ABB RAPID module: Module1.mod

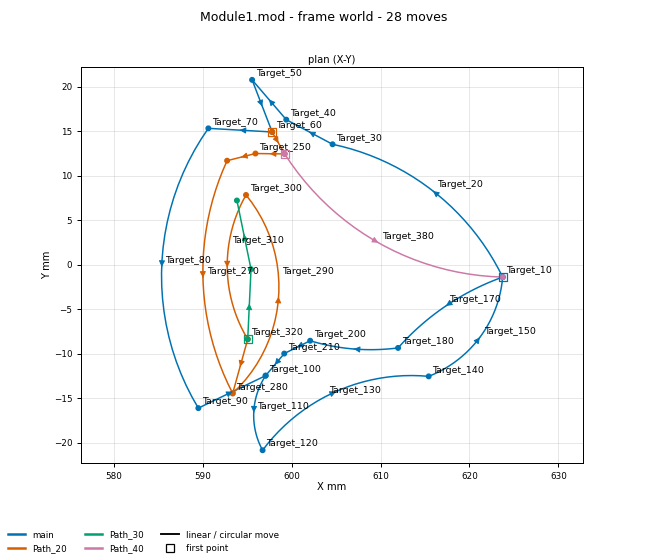
[picture p0: tool path of Module1.mod in frame world, 28 of 28 moves have a stored position in this frame; points joined in program order, loops and branches not executed]
MODULE Module1
	CONST robtarget Target_10:=[[623.736,-1.4,500],[0,0.847722968,-0.530439224,0],[-1,0,-2,0],[-1,-1,-1,-1,-1,-1]];
	CONST robtarget Target_20:=[[615.902873443,8.281748692,500],[0,0.94557602,-0.325401277,0],[0,0,-2,0],[-1,-1,-1,-1,-1,-1]];
	CONST robtarget Target_30:=[[604.61,13.532,500],[0,0.994622428,-0.103567489,0],[0,0,-2,0],[-1,-1,-1,-1,-1,-1]];
	CONST robtarget Target_40:=[[599.403600487,16.302277668,500],[0,0.943554709,-0.331216713,0],[0,0,-2,0],[-1,-1,-1,-1,-1,-1]];
	CONST robtarget Target_50:=[[595.562,20.777,500],[0,0.865930359,-0.500164587,0],[0,0,-2,0],[-1,-1,-1,-1,-1,-1]];
	CONST robtarget Target_60:=[[597.816370005,14.915141124,500],[0,0.852892303,-0.522086888,0],[0,0,-2,0],[-1,-1,-1,-1,-1,-1]];
	CONST robtarget Target_70:=[[590.643,15.324,500],[0,0.99985512,0.017021701,0],[0,0,1,0],[-1,-1,-1,-1,-1,-1]];
	CONST robtarget Target_80:=[[585.395347846,-0.237449737,500],[0,0.719631545,0.694356133,0],[-1,0,1,0],[-1,-1,-1,-1,-1,-1]];
	CONST robtarget Target_90:=[[589.518,-16.134,500],[0,0.491466316,0.870896584,0],[-1,0,0,0],[-1,-1,-1,-1,-1,-1]];
	CONST robtarget Target_100:=[[597.083,-12.483,500],[0,-0.264785252,0.964307405,0],[-1,0,-1,0],[-1,-1,-1,-1,-1,-1]];
	CONST robtarget Target_110:=[[595.746657937,-16.629604656,500],[0,0.721325087,0.69259665,0],[-1,0,1,0],[-1,-1,-1,-1,-1,-1]];
	CONST robtarget Target_120:=[[596.742,-20.871,500],[0,0.509480024,0.860482484,0],[-1,0,0,0],[-1,-1,-1,-1,-1,-1]];
	CONST robtarget Target_130:=[[603.809791295,-14.83880817,500],[0,-0.23193219,0.972731957,0],[-1,0,-1,0],[-1,-1,-1,-1,-1,-1]];
	CONST robtarget Target_140:=[[615.416517972,-12.563275607,500],[0,-0.185133559,0.982713369,0],[-1,0,-1,0],[-1,-1,-1,-1,-1,-1]];
	CONST robtarget Target_150:=[[621.175011199,-8.173115177,500],[0,-0.448574398,0.893745495,0],[-1,0,-1,0],[-1,-1,-1,-1,-1,-1]];
	CONST robtarget Target_160:=[[623.736,-1.4,500],[0,-0.677333099,0.735676473,0],[-1,0,-1,0],[-1,-1,-1,-1,-1,-1]];
	CONST robtarget Target_170:=[[617.31311623,-4.669496623,500],[0,0.926848335,0.375435965,0],[-1,0,1,0],[-1,-1,-1,-1,-1,-1]];
	CONST robtarget Target_180:=[[611.975614607,-9.363781001,500],[0,0.989682936,0.143274863,0],[-1,0,1,0],[-1,-1,-1,-1,-1,-1]];
	CONST robtarget Target_190:=[[608.374,-9.557,500],[0,0.995937158,-0.090050974,0],[-1,0,-2,0],[-1,-1,-1,-1,-1,-1]];
	CONST robtarget Target_200:=[[602.090461719,-8.557904909,500],[0,0.991973762,0.126443879,0],[-1,0,1,0],[-1,-1,-1,-1,-1,-1]];
	CONST robtarget Target_210:=[[599.177398091,-9.998243918,500],[0,0.945259462,0.326319705,0],[-1,0,1,0],[-1,-1,-1,-1,-1,-1]];
	CONST robtarget Target_220:=[[597.083,-12.483,500],[0,0.858718949,0.512446843,0],[-1,0,1,0],[-1,-1,-1,-1,-1,-1]];
	CONST robtarget Target_230:=[[597.816370005,14.915141124,500],[0,0.522086888,0.852892303,0],[0,0,0,0],[-1,-1,-1,-1,-1,-1]];
	CONST robtarget Target_240:=[[599.228158361,12.447628134,500],[0,0.481013467,0.876713205,0],[0,0,0,0],[-1,-1,-1,-1,-1,-1]];
	CONST robtarget Target_250:=[[595.93940711,12.49384908,500],[0,0.998290636,0.058444905,0],[0,0,1,0],[-1,-1,-1,-1,-1,-1]];
	CONST robtarget Target_260:=[[592.751,11.687,500],[0,0.98212196,0.18824573,0],[0,0,1,0],[-1,-1,-1,-1,-1,-1]];
	CONST robtarget Target_270:=[[590.032529197,-1.465300629,500],[0,0.698569925,0.715541794,0],[-1,0,0,0],[-1,-1,-1,-1,-1,-1]];
	CONST robtarget Target_280:=[[593.379,-14.472,500],[0,0.518908028,0.854830076,0],[-1,0,0,0],[-1,-1,-1,-1,-1,-1]];
	CONST robtarget Target_290:=[[598.550160299,-1.525622572,500],[0,0.710484728,-0.70371262,0],[-1,0,-2,0],[-1,-1,-1,-1,-1,-1]];
	CONST robtarget Target_300:=[[594.878216801,7.831632395,500],[0,0.996886245,0.078853123,0],[0,0,1,0],[-1,-1,-1,-1,-1,-1]];
	CONST robtarget Target_310:=[[592.899123752,1.965756689,500],[0,0.725029605,0.688717701,0],[0,0,1,0],[-1,-1,-1,-1,-1,-1]];
	CONST robtarget Target_320:=[[595.07,-8.388,500],[0,0.525278576,0.850930325,0],[-1,0,0,0],[-1,-1,-1,-1,-1,-1]];
	CONST robtarget Target_330:=[[593.379,-14.472,500],[0,0.825320138,0.564665096,0],[-1,0,1,0],[-1,-1,-1,-1,-1,-1]];
	CONST robtarget Target_340:=[[595.069954295,-8.387992086,500],[0,-0.64397045,0.765050364,0],[-1,0,-1,0],[-1,-1,-1,-1,-1,-1]];
	CONST robtarget Target_350:=[[595.439579744,-0.511504022,500],[0,0.734022523,-0.679125125,0],[-1,0,-2,0],[-1,-1,-1,-1,-1,-1]];
	CONST robtarget Target_360:=[[593.856,7.213,500],[0,0.812702736,-0.582678525,0],[0,0,-2,0],[-1,-1,-1,-1,-1,-1]];
	CONST robtarget Target_370:=[[599.228158361,12.447628134,500],[0,0.481013467,0.876713205,0],[0,0,0,0],[-1,-1,-1,-1,-1,-1]];
	CONST robtarget Target_380:=[[609.753497158,2.464530985,500],[0,0.254329226,0.9671177,0],[0,0,0,0],[-1,-1,-1,-1,-1,-1]];
	CONST robtarget Target_390:=[[623.736,-1.4,500],[0,0.012497461,0.999921904,0],[-1,0,0,0],[-1,-1,-1,-1,-1,-1]];
	PROC main()
	    MoveL Target_10,v1000,z0,MyNewTool\WObj:=wobj0;
	    MoveC Target_20,Target_30,v1000,z0,MyNewTool\WObj:=wobj0;
	    MoveL Target_40,v1000,z0,MyNewTool\WObj:=wobj0;
	    MoveL Target_50,v1000,z0,MyNewTool\WObj:=wobj0;
	    MoveL Target_60,v1000,z0,MyNewTool\WObj:=wobj0;
	    MoveL Target_70,v1000,z0,MyNewTool\WObj:=wobj0;
	    MoveC Target_80,Target_90,v1000,z0,MyNewTool\WObj:=wobj0;
	    MoveL Target_100,v1000,z0,MyNewTool\WObj:=wobj0;
	    MoveC Target_110,Target_120,v1000,z0,MyNewTool\WObj:=wobj0;
	    MoveC Target_130,Target_140,v1000,z0,MyNewTool\WObj:=wobj0;
	    MoveC Target_150,Target_160,v1000,z0,MyNewTool\WObj:=wobj0;
	    MoveC Target_170,Target_180,v1000,z0,MyNewTool\WObj:=wobj0;
	    MoveC Target_190,Target_200,v1000,z0,MyNewTool\WObj:=wobj0;
	    MoveL Target_210,v1000,z0,MyNewTool\WObj:=wobj0;
	    MoveL Target_220,v1000,z0,MyNewTool\WObj:=wobj0;
        Path_20;
	ENDPROC
	PROC Path_20()
	    MoveL Target_230,v1000,z0,MyNewTool\WObj:=wobj0;
	    MoveL Target_240,v1000,z0,MyNewTool\WObj:=wobj0;
	    MoveL Target_250,v1000,z0,MyNewTool\WObj:=wobj0;
	    MoveL Target_260,v1000,z0,MyNewTool\WObj:=wobj0;
	    MoveC Target_270,Target_280,v1000,z0,MyNewTool\WObj:=wobj0;
	    MoveC Target_290,Target_300,v1000,z0,MyNewTool\WObj:=wobj0;
	    MoveC Target_310,Target_320,v1000,z0,MyNewTool\WObj:=wobj0;
	    MoveL Target_330,v1000,z0,MyNewTool\WObj:=wobj0;
        Path_30;
	ENDPROC
	PROC Path_30()
	    MoveL Target_340,v1000,z0,MyNewTool\WObj:=wobj0;
	    MoveL Target_350,v1000,z0,MyNewTool\WObj:=wobj0;
	    MoveL Target_360,v1000,z0,MyNewTool\WObj:=wobj0;
        Path_40;
	ENDPROC
	PROC Path_40()
	    MoveL Target_370,v1000,z0,MyNewTool\WObj:=wobj0;
	    MoveC Target_380,Target_390,v1000,z0,MyNewTool\WObj:=wobj0;
	ENDPROC
ENDMODULE
